_CFC_ (* Continuous Function Chart, elements in execution order *)
#0 RT_VKL_OLD_SEZ_LETO:R_TRIG(CLK: TRUE)
#1 MOVE(EN: #0.Q, SCHU_P2_1_UST_SEZ_LETO)
#2 SCHU_P2_1_UST_SEZ_LETO_OLD <= #1
#3 RT_VKL_OLD_SEZ_ZIMA:R_TRIG(CLK: TRUE)
#4 MOVE(EN: #3.Q, SCHU_P2_1_UST_SEZ_ZIMA)
#5 SCHU_P2_1_UST_SEZ_ZIMA_OLD <= #4
#6 <>(SCHU_P2_1_UST_SEZ_LETO, SCHU_P2_1_UST_SEZ_LETO_OLD)
#7 >(SCHU_P2_1_UST_SEZ_LETO, SCHU_P2_1_UST_SEZ_ZIMA_OLD)
#8 AND(#6, #7)
#9 MOVE(EN: #8, SCHU_P2_1_UST_SEZ_LETO)
#10 SCHU_P2_1_UST_SEZ_LETO_OLD <= #9
#11 AND(#6, NOT #7)
#12 MOVE(EN: #11, SCHU_P2_1_UST_SEZ_LETO_OLD)
#13 SCHU_P2_1_UST_SEZ_LETO <= #12
#14 <>(SCHU_P2_1_UST_SEZ_ZIMA, SCHU_P2_1_UST_SEZ_ZIMA_OLD)
#15 <(SCHU_P2_1_UST_SEZ_ZIMA, SCHU_P2_1_UST_SEZ_LETO_OLD)
#16 AND(#14, #15)
#17 MOVE(EN: #16, SCHU_P2_1_UST_SEZ_ZIMA)
#18 SCHU_P2_1_UST_SEZ_ZIMA_OLD <= #17
#19 AND(#14, NOT #15)
#20 MOVE(EN: #19, SCHU_P2_1_UST_SEZ_ZIMA_OLD)
#21 SCHU_P2_1_UST_SEZ_ZIMA <= #20
#22 RT_UE2_VL_UST_OTKL_OLD:R_TRIG(CLK: TRUE)
#23 MOVE(EN: #22.Q, SCHU_P2_1_UE2_VL_UST_OTKL)
#24 SCHU_P2_1_UE2_VL_UST_OTKL_OLD <= #23
#25 RT_UE2_VL_UST_VKL_OLD:R_TRIG(CLK: TRUE)
#26 MOVE(EN: #25.Q, SCHU_P2_1_UE2_VL_UST_VKL)
#27 SCHU_P2_1_UE2_VL_UST_VKL_OLD <= #26
#28 <>(SCHU_P2_1_UE2_VL_UST_OTKL, SCHU_P2_1_UE2_VL_UST_OTKL_OLD)
#29 >(SCHU_P2_1_UE2_VL_UST_OTKL, SCHU_P2_1_UE2_VL_UST_VKL_OLD)
#30 AND(#28, #29)
#31 MOVE(EN: #30, SCHU_P2_1_UE2_VL_UST_OTKL)
#32 SCHU_P2_1_UE2_VL_UST_OTKL_OLD <= #31
#33 AND(#28, NOT #29)
#34 MOVE(EN: #33, SCHU_P2_1_UE2_VL_UST_OTKL_OLD)
#35 SCHU_P2_1_UE2_VL_UST_OTKL <= #34
#36 <>(SCHU_P2_1_UE2_VL_UST_VKL, SCHU_P2_1_UE2_VL_UST_VKL_OLD)
#37 <(SCHU_P2_1_UE2_VL_UST_VKL, SCHU_P2_1_UE2_VL_UST_OTKL_OLD)
#38 AND(#36, #37)
#39 MOVE(EN: #38, SCHU_P2_1_UE2_VL_UST_VKL)
#40 SCHU_P2_1_UE2_VL_UST_VKL_OLD <= #39
#41 AND(#36, NOT #37)
#42 MOVE(EN: #41, SCHU_P2_1_UE2_VL_UST_VKL_OLD)
#43 SCHU_P2_1_UE2_VL_UST_VKL <= #42
#44 RT_UE3_VL_UST_OTKL_OLD:R_TRIG(CLK: TRUE)
#45 MOVE(EN: #44.Q, SCHU_P2_1_UE3_VL_UST_OTKL)
#46 SCHU_P2_1_UE3_VL_UST_OTKL_OLD <= #45
#47 RT_UE3_VL_UST_VKL_OLD:R_TRIG(CLK: TRUE)
#48 MOVE(EN: #47.Q, SCHU_P2_1_UE3_VL_UST_VKL)
#49 SCHU_P2_1_UE3_VL_UST_VKL_OLD <= #48
#50 <>(SCHU_P2_1_UE3_VL_UST_OTKL, SCHU_P2_1_UE3_VL_UST_OTKL_OLD)
#51 >(SCHU_P2_1_UE3_VL_UST_OTKL, SCHU_P2_1_UE3_VL_UST_VKL_OLD)
#52 AND(#50, #51)
#53 MOVE(EN: #52, SCHU_P2_1_UE3_VL_UST_OTKL)
#54 SCHU_P2_1_UE3_VL_UST_OTKL_OLD <= #53
#55 AND(#50, NOT #51)
#56 MOVE(EN: #55, SCHU_P2_1_UE3_VL_UST_OTKL_OLD)
#57 SCHU_P2_1_UE3_VL_UST_OTKL <= #56
#58 <>(SCHU_P2_1_UE3_VL_UST_VKL, SCHU_P2_1_UE3_VL_UST_VKL_OLD)
#59 <(SCHU_P2_1_UE3_VL_UST_VKL, SCHU_P2_1_UE3_VL_UST_OTKL_OLD)
#60 AND(#58, #59)
#61 MOVE(EN: #60, SCHU_P2_1_UE3_VL_UST_VKL)
#62 SCHU_P2_1_UE3_VL_UST_VKL_OLD <= #61
#63 AND(#58, NOT #59)
#64 MOVE(EN: #63, SCHU_P2_1_UE3_VL_UST_VKL_OLD)
#65 SCHU_P2_1_UE3_VL_UST_VKL <= #64
#66 RT_UE3_TE_UST_VKL_OLD:R_TRIG(CLK: TRUE)
#67 MOVE(EN: #66.Q, SCHU_P2_1_UE1_T_UST)
#68 SCHU_P2_1_UE1_T_UST_OLD <= #67
#69 RT_UE2_TE_UST_OTKL_OLD:R_TRIG(CLK: TRUE)
#70 MOVE(EN: #69.Q, SCHU_P2_1_UE2_T_UST)
#71 SCHU_P2_1_UE2_T_UST_OLD <= #70
#72 RT_UE3_TE_UST_VKL_OLD:R_TRIG(CLK: TRUE)
#73 MOVE(EN: #72.Q, SCHU_P2_1_UE3_T_UST)
#74 SCHU_P2_1_UE3_T_UST_OLD <= #73
#75 <>(SCHU_P2_1_UE3_T_UST, SCHU_P2_1_UE3_T_UST_OLD)
#76 >(SCHU_P2_1_UE3_T_UST, SCHU_P2_1_UE2_T_UST_OLD)
#77 AND(#75, #76)
#78 MOVE(EN: #77, SCHU_P2_1_UE3_T_UST)
#79 SCHU_P2_1_UE3_T_UST_OLD <= #78
#80 AND(#75, NOT #76)
#81 MOVE(EN: #80, SCHU_P2_1_UE3_T_UST_OLD)
#82 SCHU_P2_1_UE3_T_UST <= #81
#83 <>(SCHU_P2_1_UE2_T_UST, SCHU_P2_1_UE2_T_UST_OLD)
#84 <(SCHU_P2_1_UE2_T_UST, SCHU_P2_1_UE3_T_UST_OLD)
#85 AND(#83, #84)
#86 MOVE(EN: #85, SCHU_P2_1_UE2_T_UST)
#87 SCHU_P2_1_UE2_T_UST_OLD <= #86
#88 AND(#83, NOT #84)
#89 MOVE(EN: #88, SCHU_P2_1_UE2_T_UST_OLD)
#90 SCHU_P2_1_UE2_T_UST <= #89
#91 <>(SCHU_P2_1_UE1_T_UST, SCHU_P2_1_UE1_T_UST_OLD)
#92 >(SCHU_P2_1_UE1_T_UST, SCHU_P2_1_UE2_T_UST_OLD)
#93 AND(#91, #92)
#94 MOVE(EN: #93, SCHU_P2_1_UE1_T_UST)
#95 SCHU_P2_1_UE1_T_UST_OLD <= #94
#96 AND(#91, NOT #92)
#97 MOVE(EN: #96, SCHU_P2_1_UE1_T_UST_OLD)
#98 SCHU_P2_1_UE1_T_UST <= #97
_END_CFC_
END_PROGRAM

(* POU Input/AI/P, CFC *)
PROGRAM P
VAR
	fb_P: ISTOK_ANALOGVH;
	ofset: REAL;
	fb_SCHU_P2_1_PE1_B_UST: ISTOK_GT;
	lor: REAL;
	highRange: REAL := 1000;		(*Максимальное показание датчика*)
	lowRange: REAL := 0;		(*Минимальное показания датчика*)
	highLimit: REAL := 1000;		(*Макасимальный уровень предупреждения*)
	lowLimit: REAL := 0;			(*Минимальный уровень предупреждения*)
END_VAR
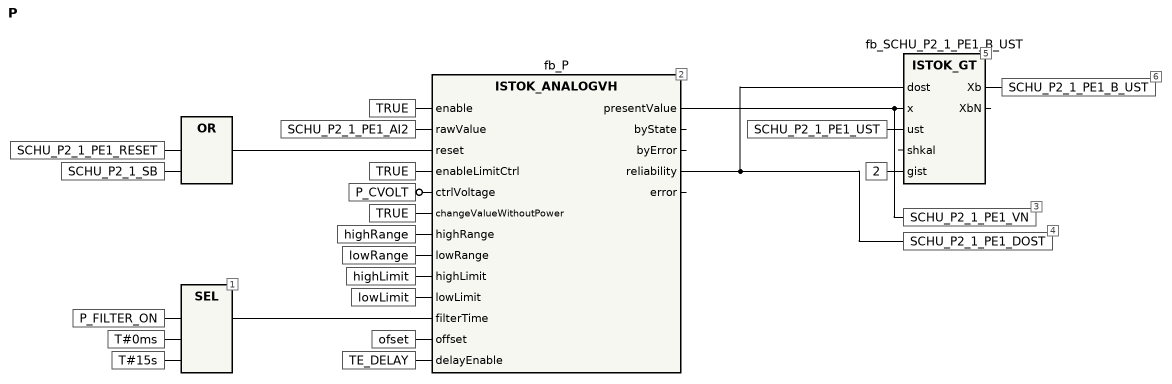
_CFC_ (* Continuous Function Chart, elements in execution order *)
#0 OR(SCHU_P2_1_PE1_RESET, SCHU_P2_1_SB)
#1 SEL(P_FILTER_ON, T#0ms, T#15s)
#2 fb_P:ISTOK_ANALOGVH(enable: TRUE, rawValue: SCHU_P2_1_PE1_AI2, reset: #0, enableLimitCtrl: TRUE, ctrlVoltage: NOT P_CVOLT, changeValueWithoutPower: TRUE, highRange: highRange, lowRange: lowRange, highLimit: highLimit, lowLimit: lowLimit, filterTime: #1, offset: ofset, delayEnable: TE_DELAY)
#3 SCHU_P2_1_PE1_VN <= #2.presentValue
#4 SCHU_P2_1_PE1_DOST <= #2.reliability
#5 fb_SCHU_P2_1_PE1_B_UST:ISTOK_GT(dost: #2.reliability, x: #2.presentValue, ust: SCHU_P2_1_PE1_UST, shkal: -, gist: 2)
#6 SCHU_P2_1_PE1_B_UST <= #5.Xb
_END_CFC_
(* the same logic as Structured Text *)
fb_P(enable := TRUE, rawValue := SCHU_P2_1_PE1_AI2, reset := SCHU_P2_1_PE1_RESET OR SCHU_P2_1_SB, enableLimitCtrl := TRUE, ctrlVoltage := NOT P_CVOLT, changeValueWithoutPower := TRUE, highRange := highRange, lowRange := lowRange, highLimit := highLimit, lowLimit := lowLimit, filterTime := SEL(P_FILTER_ON, T#0ms, T#15s), offset := ofset, delayEnable := TE_DELAY);
SCHU_P2_1_PE1_VN := fb_P.presentValue;
SCHU_P2_1_PE1_DOST := fb_P.reliability;
fb_SCHU_P2_1_PE1_B_UST(dost := fb_P.reliability, x := fb_P.presentValue, ust := SCHU_P2_1_PE1_UST, gist := 2);
SCHU_P2_1_PE1_B_UST := fb_SCHU_P2_1_PE1_B_UST.Xb;
END_PROGRAM

(* POU Lib/ISTOK_ANALOGVH, CFC *)
FUNCTION_BLOCK ISTOK_ANALOGVH
VAR_INPUT
	enable: BOOL;
	rawValue: INT;
	reset: BOOL;
	enableLimitCtrl: BOOL;
	ctrlVoltage: BOOL;
	changeValueWithoutPower: BOOL := TRUE;

	highRange: REAL;
	lowRange: REAL;
	highLimit: REAL;
	lowLimit: REAL;
	filterTime: TIME;
	offset: REAL;

	delayEnable: TIME;
END_VAR
VAR_OUTPUT
	presentValue: REAL;
	byState: BYTE;
	byError: BYTE;

	reliability: BOOL;
	error: BOOL;
END_VAR
VAR
	fb_HVACAI: FB_HVACAnalogInput;

	bEnableLimitCtrl: BOOL := TRUE;

	iHighRange: INT := 32767;
	iLowRange: INT := 0;

	tFilterTime: TIME;
	rOffset: REAL := 0;

	delay: TON;

	a: BOOL;
	b: BOOL;
	c: INT;
	d: INT;
	delay_error: TON;
	SR_AI: SR;
	RS_AI: RS;

	I_GT: ISTOK_GT;
	I_LT: ISTOK_LT;
	TON_DOST: TON;
END_VAR
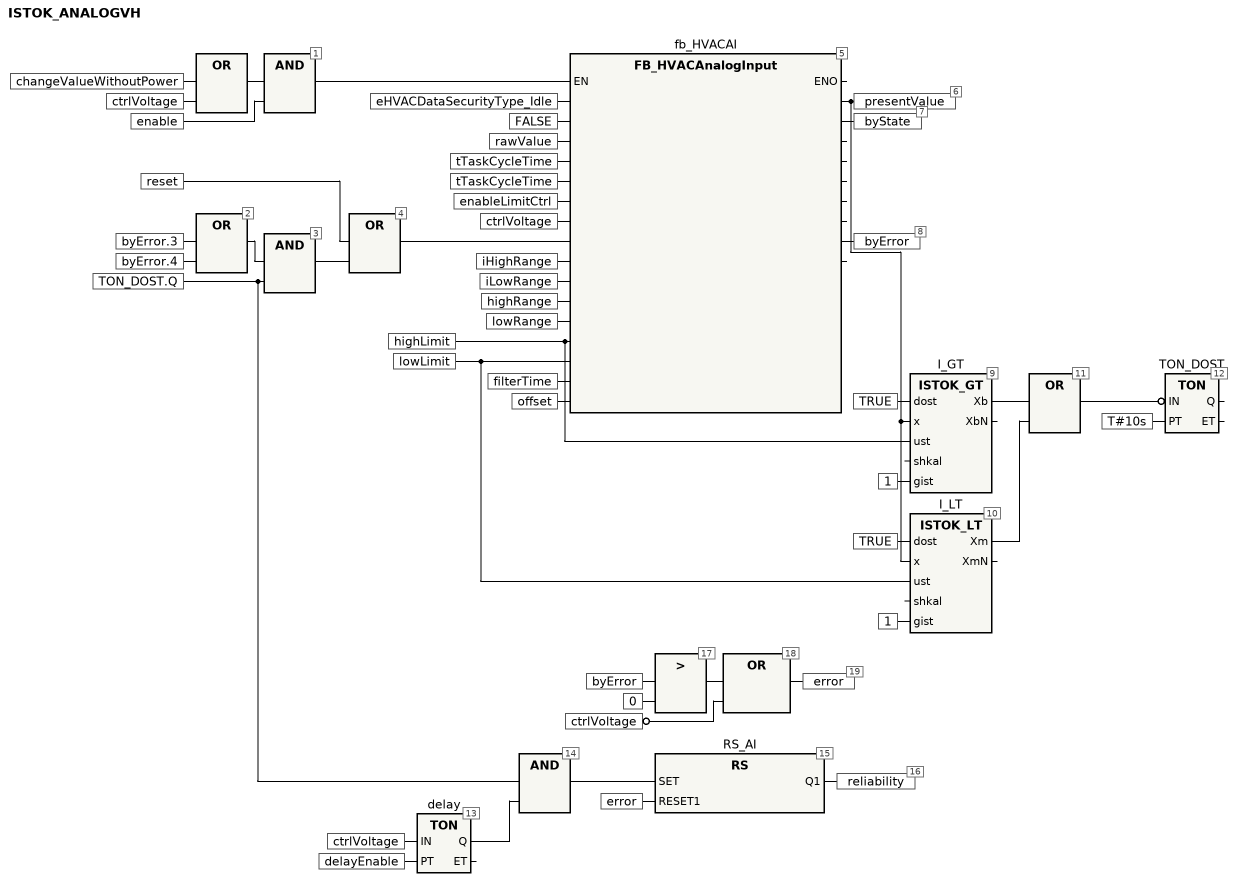
